# EPICS substitutions: epics_installer_v1.0/option/epicsIOC_musr_20221025ver/serialTestApp/Db/A100L/A100L.subs
# RAON parameters

global { CONTROLLER=musr:A100L }
file A100L.db
{ pattern
  {CH SENSOR                                         ADDR      PORT }
  { 1 "$(SENSOR1=$(P=$(CONTROLLER))"  "$(ADDR1=000)"        "$(PORT1=A100L_PORT)"}
}
